// TIA Portal V17 export
// export: Created 2023-02-26T22:59:50.6065506Z, ExportSetting WithDefaults, DisplayName Totally Integrated Automation Portal, DisplayVersion V17, DisplayName TIA Portal Openness, DisplayVersion V17, DisplayName TIA Portal Version Control Interface, DisplayVersion V17, DisplayName TIA Portal Test Suite Advanced, DisplayVersion V17, DisplayName STEP 7 Professional, DisplayVersion V17, DisplayName SIMATIC Energy Suite, DisplayVersion V17, DisplayName STEP 7 Safety, DisplayVersion V17, DisplayName WinCC Professional, DisplayVersion V17
DATA_BLOCK "LOG_LineTimeStatistic"   // DB44
{ S7_Optimized_Access := 'TRUE' }
VERSION : 0.1
// stored: AutoNumber true, IsOnlyStoredInLoadMemory false, IsRetainMemResEnabled false, IsWriteProtectedInAS false, MemoryReserve 20
   VAR RETAIN
      StartLine { S7_SetPoint := 'True'} : "stt_TimeWork";
      StopLine { S7_SetPoint := 'True'} : "stt_TimeWork";
      AutoMode { S7_SetPoint := 'True'} : "stt_TimeWork";
      ManualMode { S7_SetPoint := 'True'} : "stt_TimeWork";
      Error { S7_SetPoint := 'True'} : "stt_TimeWork";
   END_VAR
BEGIN
END_DATA_BLOCK
